% RSLogix 500 project REDES_191207_vFINAL.RSS, saved by version 12.00.00.00 %
PROJECT "UNTITLED"    % processor: Bul.1763 MicroLogix 1100 Series B %

PROGRAM FILES
  LAD 2   11 rungs

DATA FILES
  O0 OUTPUT  6 elements
  I1 INPUT  12 elements
  S2 STATUS  66 elements
  B3 BINARY  1 elements
  T4 TIMER  1 elements
  C5 COUNTER  2 elements
  R6 CONTROL  1 elements
  N7 INTEGER  100 elements
  F8 R_PHASE_F  256 elements
  MG9 MSG BLOCK  10 elements
  L10 LONG  100 elements
  N11 R_STATUS  100 elements
  N12 W_STATUS  100 elements
  F13 R_STATUS_F  80 elements
  F14 W_STATUS_F  20 elements

LADDER 2
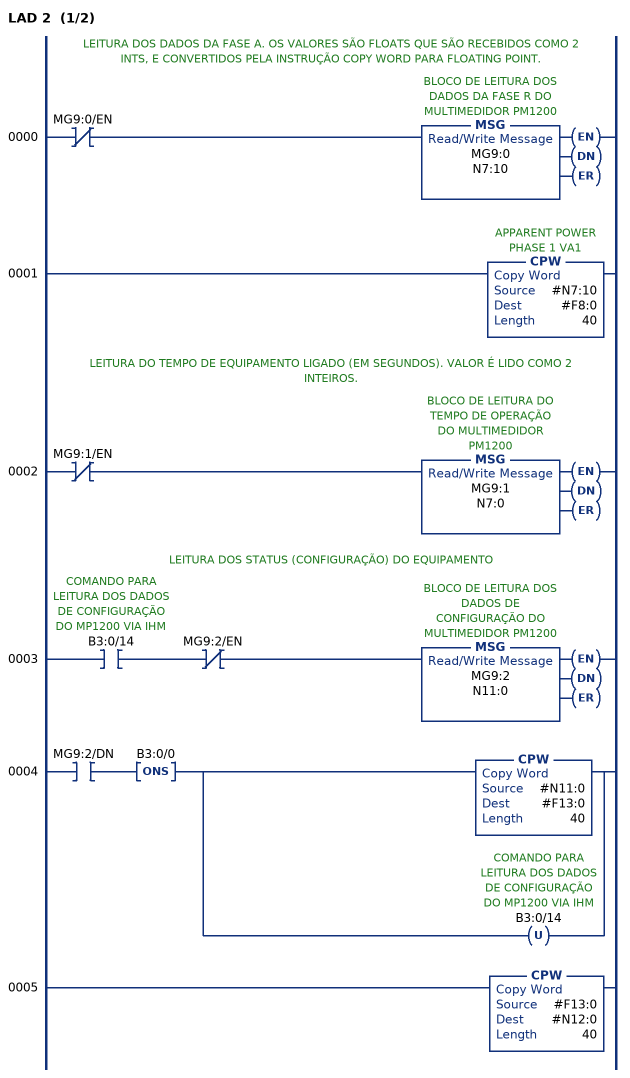
% Rung: 0 %
% LEITURA DOS DADOS DA FASE A. OS VALORES SÃO FLOATS QUE SÃO RECEBIDOS COMO 2 INTS, E CONVERTIDOS PELA INSTRUÇÃO COPY WORD PARA FLOATING POINT. %
SOR XIO MG9:0/EN MSG MG9:0 N7:10 EOR
%   MSG set-up: 03 Read Holding Registers (4xxxxx) | 10 | 20 | 3031 | N7:10 | 0 | 1 | 0 | CLIENT | 0 | 0 | ? %
%   MG9:0  "BLOCO DE LEITURA DOS DADOS DA FASE R DO MULTIMEDIDOR PM1200" %
% Rung: 1 %
SOR CPW #N7:10 #F8:0 40 EOR
%   F8:0  VA1  "APPARENT POWER PHASE 1" %
% Rung: 2 %
% LEITURA DO TEMPO DE EQUIPAMENTO LIGADO (EM SEGUNDOS). VALOR É LIDO COMO 2 INTEIROS. %
SOR XIO MG9:1/EN MSG MG9:1 N7:0 EOR
%   MSG set-up: 03 Read Holding Registers (4xxxxx) | 255 | 2 | 3993 | N7:0 | 0 | 1 | 0 | CLIENT | 0 | 0 | ? %
%   MG9:1  "BLOCO DE LEITURA DO TEMPO DE OPERAÇÃO DO MULTIMEDIDOR PM1200" %
%   N7:0  "Tempo Ligado [s] MSW" %
% Rung: 3 %
% LEITURA DOS STATUS (CONFIGURAÇÃO) DO EQUIPAMENTO %
SOR XIC B3:0/14 XIO MG9:2/EN MSG MG9:2 N11:0 EOR
%   B3:0/14  "COMANDO PARA LEITURA DOS DADOS DE CONFIGURAÇÃO DO MP1200 VIA IHM" %
%   MSG set-up: 03 Read Holding Registers (4xxxxx) | 255 | 40 | 101 | N11:0 | 0 | 1 | 0 | CLIENT | 0 | 0 | ? %
%   MG9:2  "BLOCO DE LEITURA DOS DADOS DE CONFIGURAÇÃO DO MULTIMEDIDOR PM1200" %
% Rung: 4 %
SOR XIC MG9:2/DN ONS B3:0/0 BST CPW #N11:0 #F13:0 40 NXB OTU B3:0/14 BND EOR
%   B3:0/14  "COMANDO PARA LEITURA DOS DADOS DE CONFIGURAÇÃO DO MP1200 VIA IHM" %
% Rung: 5 %
SOR CPW #F13:0 #N12:0 40 EOR

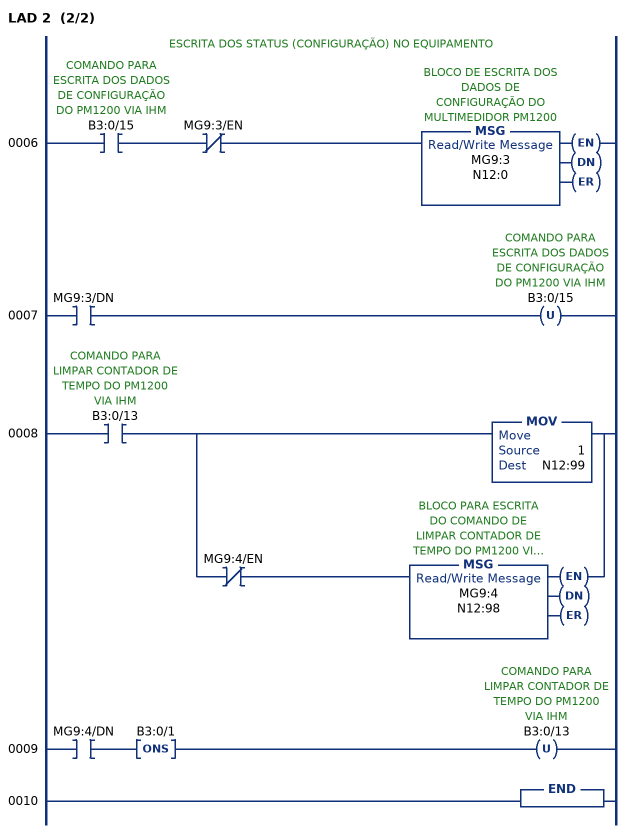
% Rung: 6 %
% ESCRITA DOS STATUS (CONFIGURAÇÃO) NO EQUIPAMENTO %
SOR XIC B3:0/15 XIO MG9:3/EN MSG MG9:3 N12:0 EOR
%   B3:0/15  "COMANDO PARA ESCRITA DOS DADOS DE CONFIGURAÇÃO DO PM1200 VIA IHM" %
%   MSG set-up: 16 Write Multiple Registers (4xxxxx) | 255 | 40 | 101 | N12:0 | 0 | 1 | 0 | CLIENT | 0 | 0 | ? %
%   MG9:3  "BLOCO DE ESCRITA DOS DADOS DE CONFIGURAÇÃO DO MULTIMEDIDOR PM1200" %
% Rung: 7 %
SOR XIC MG9:3/DN OTU B3:0/15 EOR
%   B3:0/15  "COMANDO PARA ESCRITA DOS DADOS DE CONFIGURAÇÃO DO PM1200 VIA IHM" %
% Rung: 8 %
SOR XIC B3:0/13 BST MOV 1 N12:99 NXB XIO MG9:4/EN MSG MG9:4 N12:98 BND EOR
%   B3:0/13  "COMANDO PARA LIMPAR CONTADOR DE TEMPO DO PM1200 VIA IHM" %
%   MSG set-up: 16 Write Multiple Registers (4xxxxx) | 10 | 2 | 311 | N12:98 | 0 | 1 | 0 | CLIENT | 0 | 0 | ? %
%   MG9:4  "BLOCO PARA ESCRITA DO COMANDO DE LIMPAR CONTADOR DE TEMPO DO PM1200 VIA IHM" %
% Rung: 9 %
SOR XIC MG9:4/DN ONS B3:0/1 OTU B3:0/13 EOR
%   B3:0/13  "COMANDO PARA LIMPAR CONTADOR DE TEMPO DO PM1200 VIA IHM" %
% Rung: 10 %
SOR END EOR

OTHER DOCUMENTED ADDRESSES
  B3:1  "ALWAYS ON"
  F8:1  W1  "ACTIVE POWER PHASE 1"
  F8:2  VAR1  "REACTIVE POWER PHASE 1"
  F8:3  PF1  "POWER FACTOR PHASE 1"
  F8:4  V12  "VOLTAGE PHASE 1 TO PHASE 2"
  F8:5  V1  "VOLTAGE PHASE 1 TO NEUTRAL"
  F8:6  A1  "CURRENT PHASE 1"
  F8:7  F1  "FREQUENCY PHASE 1 [Hz]"
  F8:8  "RESERVED"
  F8:9  INTER1  "NUMBER OF INTERRUPTION"
  F8:180  "TESTE V_PRI ESCRITA"
  MG9:0.16/15  "BLOCO DE LEITURA DOS DADOS DA FASE R DO MULTIMEDIDOR PM1200 MSG HABILITADO"
  MG9:1.16/15  "BLOCO DE LEITURA DO TEMPO DE OPERAÇÃO DO MULTIMEDIDOR PM1200 MSG HABILITADO"
  MG9:2.16/15  "BLOCO DE LEITURA DOS DADOS DE CONFIGURAÇÃO DO MULTIMEDIDOR PM1200 MSG HABILITADO"
  MG9:2.17/13  "BLOCO DE LEITURA DOS DADOS DE CONFIGURAÇÃO DO MULTIMEDIDOR PM1200 MSG CONCLUÍDO"
  MG9:3.16/15  "BLOCO DE ESCRITA DOS DADOS DE CONFIGURAÇÃO DO MULTIMEDIDOR PM1200 MSG HABILITADO"
  MG9:3.17/13  "BLOCO DE ESCRITA DOS DADOS DE CONFIGURAÇÃO DO MULTIMEDIDOR PM1200 MSG CONCLUÍDO"
  N7:1  "Tempo Ligado [s] LSW"

COMMENTS NOT ATTACHED TO A CURRENT RUNG
  L10:0: JUNTA OS DOIS INTEIROS EM UM LONG
  MG9:1: LEITURA DO TEMPO DE EQUIPAMENTO LIGADO (EM SEGUNDOS). VALOR É LIDO COMO 2 INTEIROS.
  MG9:0: LEITURA DA TENSÃO FASE-NEUTRO PARA FASE A. O VALOR É UM FLOAT QUE É LIDO COMO 2 INT, E CONVERTIDO PELA INSTRUÇÃO COPY WORD PARA FLOATING POINT.

DATA TABLE (non-zero values as saved)
DATA B3
% B3:0 % 0X0003
DATA C5
% .PRE .ACC %
% C5:0 % 100 37
DATA N7
% N7:0 % 0 242 0 0 0 0 0 0 0 0
% N7:10 % 0 0 23691 9321 23691 9321 -27921 8595 23589 8533
% N7:20 % -8363 17081 26763 9377 7960 17008 1 9257 0 0
DATA F8
% F8:0 % 0 5.060221e-17 5.060221e-17 1e-18 7.228916e-19
% F8:5 % 92.9362 6.999972e-17 60.03036 3.664604e-17 0
% F8:180 % 300 0 0 0 0
DATA L10
% L10:0 % 12176 0 0 0 0
DATA N11
% N11:0 % 0 17327 42 16544 0 17302 -32768 17359 0 16576
% N11:10 % 0 16256 0 0 0 16256 0 16384 0 16448
% N11:20 % 0 16544 0 0 0 16256 0 17096 0 16384
% N11:30 % 0 16384 0 17530 0 16384 -4096 17792 -10486 15267
DATA N12
% N12:0 % 0 17327 42 16544 0 17302 -32768 17359 0 16576
% N12:10 % 0 16256 0 0 0 16256 0 16384 0 16448
% N12:20 % 0 16544 0 0 0 16256 0 17096 0 16384
% N12:30 % 0 16384 0 17530 0 16384 -4096 17792 -10486 15267
% N12:90 % 0 0 0 0 0 0 0 0 0 1
DATA F13
% F13:0 % 350 5.00002 300 415 6
% F13:5 % 1 0 1 2 3
% F13:10 % 5 0 1 100 2
% F13:15 % 2 1000 2 4126 0.005
